Omron CX-Programmer project NewProject (CX-Programmer 9.61)

# PLC AutomaticConveyorSystem: CJ2M CPU11

## Global symbols (name address type ; comment)
0 CHANNEL  ; Object_A
0.00 BOOL  ; Start_button
0.01 BOOL  ; Emergency_Button
0.02 BOOL  ; Color_Sensor_A
0.03 BOOL  ; Color_Sensor_B
0.04 BOOL  ; Proximity_Sensor
0.05 BOOL  ; Manual
0.06 BOOL  ; P_Conveyor
0.07 BOOL  ; P_Solenoid_A
0.08 BOOL  ; P_Solenoid_B
0.09 BOOL  ; Reset
100.00 BOOL  ; Start
100.01 BOOL  ; Conveyor
100.02 BOOL  ; Solenoid_A
100.03 BOOL  ; Solenoid_B
C0000 BOOL  ; Object_B
D100 CHANNEL  ; Total_A
D200 CHANNEL  ; Total_B

## Program NewProgram1 (cyclic task 0)

### Section Section1

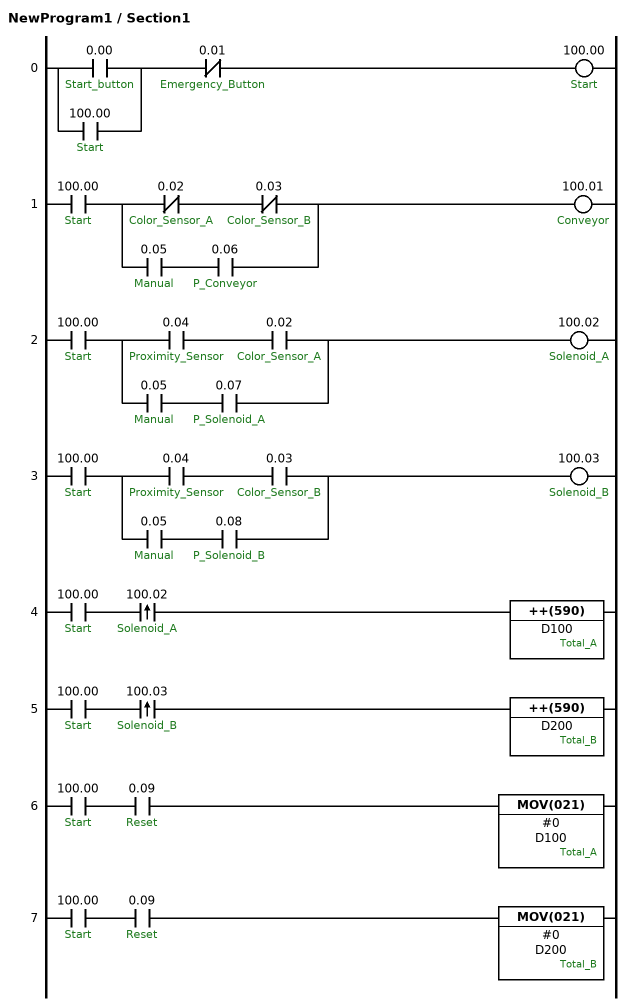
; rung 0
LD 0.00  ; Start_button
OR 100.00  ; Start
ANDNOT 0.01  ; Emergency_Button
OUT 100.00  ; Start
; rung 1
LD 100.00  ; Start
LDNOT 0.02  ; Color_Sensor_A
ANDNOT 0.03  ; Color_Sensor_B
LD 0.05  ; Manual
AND 0.06  ; P_Conveyor
ORLD
ANDLD
OUT 100.01  ; Conveyor
; rung 2
LD 100.00  ; Start
LD 0.04  ; Proximity_Sensor
AND 0.02  ; Color_Sensor_A
LD 0.05  ; Manual
AND 0.07  ; P_Solenoid_A
ORLD
ANDLD
OUT 100.02  ; Solenoid_A
; rung 3
LD 100.00  ; Start
LD 0.04  ; Proximity_Sensor
AND 0.03  ; Color_Sensor_B
LD 0.05  ; Manual
AND 0.08  ; P_Solenoid_B
ORLD
ANDLD
OUT 100.03  ; Solenoid_B
; rung 4
LD 100.00  ; Start
@AND 100.02  ; Solenoid_A
++(590) D100  ; Total_A
; rung 5
LD 100.00  ; Start
@AND 100.03  ; Solenoid_B
++(590) D200  ; Total_B
; rung 6
LD 100.00  ; Start
AND 0.09  ; Reset
MOV(021) #0 D100  ; Total_A
; rung 7
LD 100.00  ; Start
AND 0.09  ; Reset
MOV(021) #0 D200  ; Total_B

### Section END
; rung 0
END(001)